// TIA Portal V20 export
FUNCTION_BLOCK "FB_DigitalOutputs"   // FB212, SCL
{ S7_Optimized_Access := 'TRUE' }
// stored: AutoNumber false, MemoryReserve 100, SetENOAutomatically false
   VAR
      sFreeQ0_0 : "FB_DigitalOutput";
      sOperatingCounter : "FB_DigitalOutput";
      sGeneralAirValve : "FB_DigitalOutput";
      sSmartLineDisable : "FB_DigitalOutput";
      sMachineLight : "FB_DigitalOutput";
      sMachineLightBack : "FB_DigitalOutput";
      sLightTowerOrange : "FB_DigitalOutput";
      sLightTowerRed : "FB_DigitalOutput";
      sLightTowerBlue : "FB_DigitalOutput";
      sLightTowerGreen : "FB_DigitalOutput";
      sLightTowerWhite : "FB_DigitalOutput";
      sBacklight : "FB_DigitalOutput";
      sFreeQ1_4 : "FB_DigitalOutput";
      sInfeedON : "FB_DigitalOutput";
      sAxisActivation : "FB_DigitalOutput";
      sBuzzerActivation : "FB_DigitalOutput";
      sElbaronPowerON : "FB_DigitalOutput";
      sObservationCameraLight : "FB_DigitalOutput";
      sLaserExternalDoorOpening : "FB_DigitalOutput";
      sCoolingStart : "FB_DigitalOutput";
      sX_AxisBrakeActivation : "FB_DigitalOutput";
      sY_AxisBrakeActivation : "FB_DigitalOutput";
      sAxisB_TeachInClampingPart : "FB_DigitalOutput";
      sEPO_UPS : "FB_DigitalOutput";
      sHeadLaserStart : "FB_DigitalOutput";
      sHeadLaserStop : "FB_DigitalOutput";
      sAxis2_PowerContactor : "FB_DigitalOutput";
      sGasAssistOn : "FB_DigitalOutput";
      sSmartLineReset : "FB_DigitalOutput";
      sXY_AxisPowerContactor : "FB_DigitalOutput";
      sLaserAirPressureProcess : "FB_DigitalOutput";
      sBus60V_PowerContactor : "FB_DigitalOutput";
      sFreeQ4_0 : "FB_DigitalOutput";
      sFreeQ4_1 : "FB_DigitalOutput";
      sFreeQ4_2 : "FB_DigitalOutput";
      sFreeQ4_3 : "FB_DigitalOutput";
      sLoadClampClosing : "FB_DigitalOutput";
      sLoadClampOpening : "FB_DigitalOutput";
      sUnloadClampClosing : "FB_DigitalOutput";
      sUnloadClampOpening : "FB_DigitalOutput";
      sClampingOpening : "FB_DigitalOutput";
      sClampingClosing : "FB_DigitalOutput";
      sB_AxisBrakeRelease : "FB_DigitalOutput";
      sSuction : "FB_DigitalOutput";
      sFreeQ5_4 : "FB_DigitalOutput";
      sFreeQ5_5 : "FB_DigitalOutput";
      sFreeQ5_6 : "FB_DigitalOutput";
      sFreeQ5_7 : "FB_DigitalOutput";
      sExternalGateClosing : "FB_DigitalOutput";
      sExternalGateOpening : "FB_DigitalOutput";
      sInternalGateClosing : "FB_DigitalOutput";
      sInternalGateOpening : "FB_DigitalOutput";
      sPowerMeterRetract : "FB_DigitalOutput";
      sPowerMeterAdvance : "FB_DigitalOutput";
      sBlowing : "FB_DigitalOutput";
      sFreeQ8_7 : "FB_DigitalOutput";
      sFreeQ9_0 : "FB_DigitalOutput";
      sFreeQ9_1 : "FB_DigitalOutput";
      sFreeQ9_2 : "FB_DigitalOutput";
      sFreeQ9_3 : "FB_DigitalOutput";
      sFreeQ9_4 : "FB_DigitalOutput";
      sFreeQ9_5 : "FB_DigitalOutput";
      sFreeQ9_6 : "FB_DigitalOutput";
      sFreeQ9_7 : "FB_DigitalOutput";
      sSonplasDiagDPCoupler { S7_SetPoint := 'True'} : "FB_DigitalOutput";
      sSonplasReady { S7_SetPoint := 'True'} : "FB_DigitalOutput";
      sSonplasNoEStop { S7_SetPoint := 'True'} : "FB_DigitalOutput";
      sSonplasDoorsClosed { S7_SetPoint := 'True'} : "FB_DigitalOutput";
      sSonplasRunError { S7_SetPoint := 'True'} : "FB_DigitalOutput";
      sSonplasFreeQ200_5 { S7_SetPoint := 'True'} : "FB_DigitalOutput";
      sSonplasFreeQ200_6 { S7_SetPoint := 'True'} : "FB_DigitalOutput";
      sSonplasFreeQ200_7 { S7_SetPoint := 'True'} : "FB_DigitalOutput";
      sSonplasFreeQ201_0 { S7_SetPoint := 'True'} : "FB_DigitalOutput";
      sSonplasFreeQ201_1 { S7_SetPoint := 'True'} : "FB_DigitalOutput";
      sSonplasFreeQ201_2 { S7_SetPoint := 'True'} : "FB_DigitalOutput";
      sSonplasFreeQ201_3 { S7_SetPoint := 'True'} : "FB_DigitalOutput";
      sSonplasFreeQ201_4 { S7_SetPoint := 'True'} : "FB_DigitalOutput";
      sSonplasFreeQ201_5 { S7_SetPoint := 'True'} : "FB_DigitalOutput";
      sSonplasFreeQ201_6 { S7_SetPoint := 'True'} : "FB_DigitalOutput";
      sSonplasFreeQ201_7 { S7_SetPoint := 'True'} : "FB_DigitalOutput";
      sSonplasShuttle1InPos { S7_SetPoint := 'True'} : "FB_DigitalOutput";
      sSonplasFreeQ202_1 { S7_SetPoint := 'True'} : "FB_DigitalOutput";
      sSonplasFreeQ202_2 { S7_SetPoint := 'True'} : "FB_DigitalOutput";
      sSonplasFreeQ202_3 { S7_SetPoint := 'True'} : "FB_DigitalOutput";
      sSonplasFreeQ202_4 { S7_SetPoint := 'True'} : "FB_DigitalOutput";
      sSonplasFreeQ202_5 { S7_SetPoint := 'True'} : "FB_DigitalOutput";
      sSonplasPart1OK { S7_SetPoint := 'True'} : "FB_DigitalOutput";
      sSonplasPart1NOK { S7_SetPoint := 'True'} : "FB_DigitalOutput";
      sSonplasShuttle2InPos { S7_SetPoint := 'True'} : "FB_DigitalOutput";
      sSonplasFreeQ203_1 { S7_SetPoint := 'True'} : "FB_DigitalOutput";
      sSonplasFreeQ203_2 { S7_SetPoint := 'True'} : "FB_DigitalOutput";
      sSonplasFreeQ203_3 { S7_SetPoint := 'True'} : "FB_DigitalOutput";
      sSonplasFreeQ203_4 { S7_SetPoint := 'True'} : "FB_DigitalOutput";
      sSonplasFreeQ203_5 { S7_SetPoint := 'True'} : "FB_DigitalOutput";
      sSonplasPart2OK { S7_SetPoint := 'True'} : "FB_DigitalOutput";
      sSonplasPart2NOK { S7_SetPoint := 'True'} : "FB_DigitalOutput";
      sSonplasResultAccepted { S7_SetPoint := 'True'} : "FB_DigitalOutput";
      sSonplasFreeQ244_1 { S7_SetPoint := 'True'} : "FB_DigitalOutput";
      sSonplasFreeQ244_2 { S7_SetPoint := 'True'} : "FB_DigitalOutput";
      sSonplasFreeQ244_3 { S7_SetPoint := 'True'} : "FB_DigitalOutput";
      sSonplasFreeQ244_4 { S7_SetPoint := 'True'} : "FB_DigitalOutput";
      sSonplasFreeQ244_5 { S7_SetPoint := 'True'} : "FB_DigitalOutput";
      sSonplasFreeQ244_6 { S7_SetPoint := 'True'} : "FB_DigitalOutput";
      sSonplasFreeQ244_7 { S7_SetPoint := 'True'} : "FB_DigitalOutput";
   END_VAR
BEGIN
   REGION Description head
       //==================================================================================
       // POSALUX Swiss SA / (C) Copyright 2025
       //----------------------------------------------------------------------------------
       // Title: Digital Ouputs mapping
       // Comment/Function: Digital Ouputs mapping
       // Author: Fabien WALDT
       // Engineering: TIA Portal v17
       //----------------------------------------------------------------------------------
       // Change log table:
       // Version  | Date     | Expert in charge | Changes applied
       //----------------------------------------------------------------------------------
       // 00.00.01 | 20250423 | WFA              | First released version
       //==================================================================================
   END_REGION


       // ET200SP Mapping
   REGION Q0.0 - Q1.7 : DQ 16x24VDC/0.5A ST Slot 5
       #sFreeQ0_0(oHWStatus => "DQ_FreeQ0_0");
       #sOperatingCounter(oHWStatus => "DQ_OperatingCounter");
       #sGeneralAirValve(oHWStatus => "DQ_GeneralAirValve");
       #sSmartLineDisable(oHWStatus => "DQ_SmartLineDisable");
       #sMachineLight(oHWStatus => "DQ_MachineLight");
       #sMachineLightBack(oHWStatus => "DQ_MachineLightBack");
       #sLightTowerOrange(oHWStatus => "DQ_LightTowerOrange");
       #sLightTowerRed(oHWStatus => "DQ_LightTowerRed");
       //
       #sLightTowerBlue(oHWStatus => "DQ_LightTowerBlue");
       #sLightTowerGreen(oHWStatus => "DQ_Light_owerGreen");
       #sLightTowerWhite(oHWStatus => "DQ_LightTowerWhite");
       #sBacklight(oHWStatus => "DQ_Backlight");
       #sFreeQ1_4(oHWStatus => "DQ_FreeQ1_4");
       #sInfeedON(oHWStatus => "DQ_InfeedON");
       #sAxisActivation(oHWStatus => "DQ_AxisActivation");
       #sBuzzerActivation(oHWStatus => "DQ_BuzzerActivation");
   END_REGION

   REGION Q2.0 - Q3.7 : DQ 16x24VDC/0.5A ST Slot 6
       #sElbaronPowerON(oHWStatus => "DQ_ElbaronPowerON");
       #sObservationCameraLight(oHWStatus => "DQ_ObservationCameraLight");
       #sLaserExternalDoorOpening(oHWStatus => "DQ_LaserExternalDoorOpening");
       #sCoolingStart(oHWStatus => "DQ_CoolingStart");
       #sX_AxisBrakeActivation(oHWStatus => "DQ_X_AxisBrakeActivation");
       #sY_AxisBrakeActivation(oHWStatus => "DQ_Y_AxisBrakeActivation");
       #sAxisB_TeachInClampingPart(oHWStatus => "DQ_AxisB_TeachInClampingPart");
       #sEPO_UPS(oHWStatus => "DQ_EPO_UPS");
       //
       #sHeadLaserStart(oHWStatus => "DQ_HeadLaserStart");
       #sHeadLaserStop(oHWStatus => "DQ_HeadLaserStop");
       #sAxis2_PowerContactor(oHWStatus => "DQ_Axis2_PowerContactor");
       #sGasAssistOn(oHWStatus => "DQ_GasAssistOn");
       #sSmartLineReset(oHWStatus => "DQ_SmartLineReset");
       #sXY_AxisPowerContactor(oHWStatus => "DQ_XY_AxisPowerContactor");
       #sLaserAirPressureProcess(oHWStatus => "DQ_LaserAirPressureProcess");
       #sBus60V_PowerContactor(oHWStatus => "DQ_Bus60V_PowerContactor");
   END_REGION

   REGION Q4.0 - Q5.7 : DQ 16x24VDC/0.5A ST Slot 7
       #sFreeQ4_0(oHWStatus => "DQ_FreeQ4_0");
       #sFreeQ4_1(oHWStatus => "DQ_FreeQ4_1");
       #sFreeQ4_2(oHWStatus => "DQ_FreeQ4_2");
       #sFreeQ4_3(oHWStatus => "DQ_FreeQ4_3");
       #sLoadClampClosing(oHWStatus => "DQ_LoadClampClosing");
       #sLoadClampOpening(oHWStatus => "DQ_LoadClampOpening");
       #sUnloadClampClosing(oHWStatus => "DQ_UnloadClampClosing");
       #sUnloadClampOpening(oHWStatus => "DQ_UnloadClampOpening");
       //
       #sClampingOpening(oHWStatus => "DQ_ClampingOpening");
       #sClampingClosing(oHWStatus => "DQ_ClampingClosing");
       #sB_AxisBrakeRelease(oHWStatus => "DQ_B_AxisBrakeRelease");
       #sSuction(oHWStatus => "DQ_Suction");
       #sFreeQ5_4(oHWStatus => "DQ_FreeQ5_4");
       #sFreeQ5_5(oHWStatus => "DQ_FreeQ5_5");
       #sFreeQ5_6(oHWStatus => "DQ_FreeQ5_6");
       #sFreeQ5_7(oHWStatus => "DQ_FreeQ5_7");
   END_REGION

   REGION Q8.0 - Q9.7 : DQ 16x24VDC/0.5A ST Slot 8
       #sExternalGateClosing(oHWStatus => "DQ_ExternalGateClosing");
       #sExternalGateOpening(oHWStatus => "DQ_ExternalGateOpening");
       #sInternalGateClosing(oHWStatus => "DQ_InternalGateClosing");
       #sInternalGateOpening(oHWStatus => "DQ_InternalGateOpening");
       #sPowerMeterRetract(oHWStatus => "DQ_PowerMeterRetract");
       #sPowerMeterAdvance(oHWStatus => "DQ_PowerMeterAdvance");
       #sBlowing(oHWStatus => "DQ_Blowing");
       #sFreeQ8_7(oHWStatus => "DQ_FreeQ8_7");
       //
       #sFreeQ9_0(oHWStatus => "DQ_FreeQ9_0");
       #sFreeQ9_1(oHWStatus => "DQ_FreeQ9_1");
       #sFreeQ9_2(oHWStatus => "DQ_FreeQ9_2");
       #sFreeQ9_3(oHWStatus => "DQ_FreeQ9_3");
       #sFreeQ9_4(oHWStatus => "DQ_FreeQ9_4");
       #sFreeQ9_5(oHWStatus => "DQ_FreeQ9_5");
       #sFreeQ9_6(oHWStatus => "DQ_FreeQ9_6");
       #sFreeQ9_7(oHWStatus => "DQ_FreeQ9_7");
   END_REGION
END_FUNCTION_BLOCK
